// TIA Portal project "AutoII-G1" (V16)

(* hardware
DEVICE "S7-1200 station_1"  S7-1200 Station
   slot 0: "Rack_0"  S7-1200 Rack  Rack  V1.0
   slot 1: "PLC_1"  CPU 1214C DC/DC/DC  6ES7 214-1AG40-0XB0  V4.4
   slot 2: "DI 16/DQ 16x24VDC_1"  6ES7 223-1BL32-0XB0  V2.0
DEVICE "HMI_1"  KTP700 Basic PN
   slot 0: "HMI_1"  KTP700 Basic PN  6AV2 123-2GB03-0AX0  16.0.0.0
   slot 1: "HMI_RT_1"  KTP700 Basic PN  6AV2 123-2GB03-0AX0  16.0.0.0
   slot 5: "HMI_1.IE_CP_1"  PROFINET Interface  16.0.0.0
      slot 1: "Interfaz PROFINET_1"  PROFINET Interface
         slot 1: "Port_1"  Port
*)

// ===== PLC "PLC_1"  CPU 1214C DC/DC/DC =====

VAR_GLOBAL   // PLC tag table "Tabla de variables estándar"
   "ARRANQUE_M1" AT %I0.0 : Bool;
   "PARO_M1" AT %I0.1 : Bool;
   "FALLA_M1" AT %I0.2 : Bool;
   "MOTOR1" AT %Q0.0 : Bool;
   "ARRANQUE_M2" AT %I0.3 : Bool;
   "PARO_M2" AT %I0.4 : Bool;
   "FALLA_M2" AT %I0.5 : Bool;
   "MOTOR2" AT %Q0.1 : Bool;
   "ARRANQUE_M3" AT %I0.6 : Bool;
   "PARO_M3" AT %I0.7 : Bool;
   "FALLA_M3" AT %I1.0 : Bool;
   "MOTOR3" AT %Q0.2 : Bool;
   "Tag_1" AT %M0.0 : Bool;
   "Tag_2" AT %M0.1 : Bool;
   "Tag_3" AT %M0.2 : Bool;
   "Abrir_V1" AT %I2.0 : Bool;
   "Cerrar_V1" AT %I2.1 : Bool;
   "Q_Abrir_V1" AT %Q2.0 : Bool;
   "Aux_V1" AT %M2.0 : Bool;
   "Tag_4" AT %Q0.3 : Bool;
   "Conf_Ab_V1" AT %I2.2 : Bool;
   "Conf_Cer_V1" AT %I2.3 : Bool;
   "Q_Cerrar_V1" AT %Q2.1 : Bool;
   "HMI_Arranque_Secuencia" AT %M1.0 : Bool;
   "HMI_Paro_Secuencia" AT %M1.1 : Bool;
   "Reset_Fallas" AT %I2.4 : Bool;
   "Alarmas_1" AT %MW10 : Word;
   "Tag_5" AT %I3.0 : Bool;
   "Tag_6" AT %I3.1 : Bool;
   "Tag_7" AT %I3.3 : Bool;
   "Tag_8" AT %I3.2 : Bool;
   "Tag_9" AT %Q3.0 : Bool;
   "Tag_10" AT %Q3.1 : Bool;
   "Tag_11" AT %I4.0 : Bool;
   "Tag_12" AT %I4.1 : Bool;
   "Tag_13" AT %Q4.0 : Bool;
   "Tag_14" AT %Q4.1 : Bool;
   "LT-T001" AT %MD20 : Real;
   "SEÑAL T001" AT %MW18 : Int;
END_VAR

DATA_BLOCK "VALVULA_V1"   // DB3
{ S7_Optimized_Access := 'TRUE' }
VERSION : 0.1
// stored: InstanceOfName VALVULA
"VALVULA"
BEGIN
END_DATA_BLOCK

DATA_BLOCK "VALVULA_2"   // DB4
{ S7_Optimized_Access := 'TRUE' }
VERSION : 0.1
// stored: InstanceOfName VALVULA
"VALVULA"
BEGIN
END_DATA_BLOCK

DATA_BLOCK "VALVULA_3"   // DB5
{ S7_Optimized_Access := 'TRUE' }
VERSION : 0.1
// stored: InstanceOfName VALVULA
"VALVULA"
BEGIN
END_DATA_BLOCK

// folder: System blocks/Program resources

DATA_BLOCK "T_ON_M2"   // DB1
{ S7_Optimized_Access := 'TRUE' }
AUTHOR : Simatic
FAMILY : IEC
NAME : IEC_TMR
VERSION : 1.0
// stored: InstanceOfName IEC_TIMER
"IEC_TIMER"
BEGIN
END_DATA_BLOCK

DATA_BLOCK "T_ON_M3"   // DB2
{ S7_Optimized_Access := 'TRUE' }
AUTHOR : Simatic
FAMILY : IEC
NAME : IEC_TMR
VERSION : 1.0
// stored: InstanceOfName IEC_TIMER
"IEC_TIMER"
BEGIN
END_DATA_BLOCK

// folder: (top level)

FUNCTION_BLOCK "VALVULA"   // FB1, LAD
{ S7_Optimized_Access := 'TRUE' }
VERSION : 0.1
   VAR_INPUT
      Abrir : Bool;
      Conf_Abierta : Bool;
      Hab_Conf_Ab : Bool;
      T_Abrir : Time;
      T_Mon_Abrir : Time;
      Cerrar : Bool;
      Conf_Cerrada : Bool;
      Hab_Conf_Cer : Bool;
      T_Cierre : Time;
      T_Mon_Cierre : Time;
      Reset : Bool;
   END_VAR
   VAR_OUTPUT
      Q_Abrir : Bool;
      Q_Cerrar : Bool;
      Error_Abrir : Bool;
      Error_Cerrar : Bool;
   END_VAR
   VAR
      Aux_Valvula : Bool;
      Aux_Valvula2 : Bool;
      TP_Cierre : IEC_TIMER;
      TP_Abrir : IEC_TIMER;
      Mon_Abrir : IEC_TIMER;
      Mon_Cerrar : IEC_TIMER;
   END_VAR
BEGIN

REGION Network 1
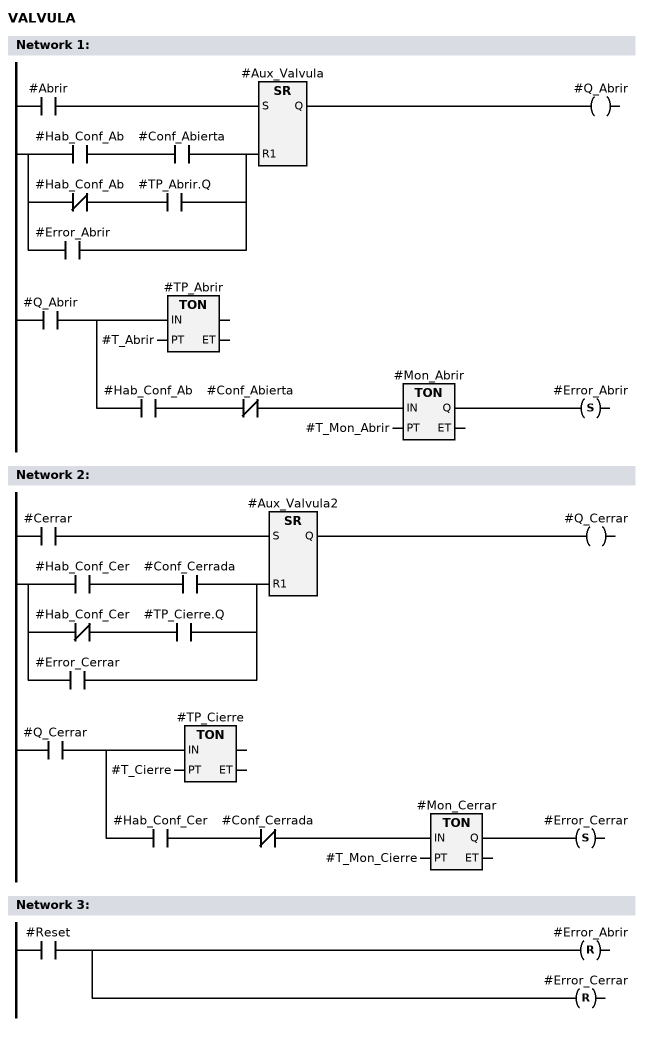
   IF #Abrir THEN
       #Aux_Valvula := TRUE;   // SR flip-flop
   END_IF;
   IF (#Hab_Conf_Ab AND #Conf_Abierta) OR (NOT #Hab_Conf_Ab AND #TP_Abrir.Q) OR #Error_Abrir THEN
       #Aux_Valvula := FALSE;
   END_IF;
   #Q_Abrir := #Aux_Valvula;
   #TP_Abrir.TON(IN := #Q_Abrir, PT := #T_Abrir);
   #Mon_Abrir.TON(IN := #Q_Abrir AND #Hab_Conf_Ab AND NOT #Conf_Abierta, PT := #T_Mon_Abrir);
   IF #Mon_Abrir.Q THEN #Error_Abrir := TRUE; END_IF;
END_REGION

REGION Network 2
   IF #Cerrar THEN
       #Aux_Valvula2 := TRUE;   // SR flip-flop
   END_IF;
   IF (#Hab_Conf_Cer AND #Conf_Cerrada) OR (NOT #Hab_Conf_Cer AND #TP_Cierre.Q) OR #Error_Cerrar THEN
       #Aux_Valvula2 := FALSE;
   END_IF;
   #Q_Cerrar := #Aux_Valvula2;
   #TP_Cierre.TON(IN := #Q_Cerrar, PT := #T_Cierre);
   #Mon_Cerrar.TON(IN := #Q_Cerrar AND #Hab_Conf_Cer AND NOT #Conf_Cerrada, PT := #T_Mon_Cierre);
   IF #Mon_Cerrar.Q THEN #Error_Cerrar := TRUE; END_IF;
END_REGION

REGION Network 3
   RUNG wire#powerrail
      Contact( #Reset )
      wire#w1
      R_Coil( #Error_Abrir )
   END_RUNG
   RUNG wire#w1
      R_Coil( #Error_Cerrar )
   END_RUNG
   // the same network as SCL:
   IF #Reset THEN
       #Error_Abrir := FALSE;
       #Error_Cerrar := FALSE;
   END_IF;
END_REGION
END_FUNCTION_BLOCK

FUNCTION "MOTOR" : Void   // FC1, LAD
{ S7_Optimized_Access := 'TRUE' }
VERSION : 0.1
   VAR_INPUT
      ARRANQUE : Bool;
      PARO : Bool;
      FALLA : Bool;
   END_VAR
   VAR_OUTPUT
      MOTOR : Bool;
   END_VAR
   VAR_IN_OUT
      mARRANQUE : Bool;
   END_VAR
BEGIN

REGION Network 1
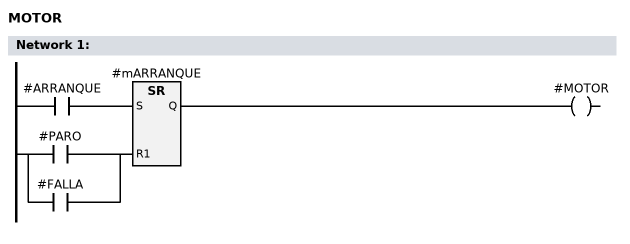
   RUNG wire#powerrail
      Contact( #ARRANQUE )
      S_SR(operand := #mARRANQUE, r1 := wire#w1)
      Coil( #MOTOR )
   END_RUNG
   RUNG wire#powerrail
      Contact( #PARO )
   END_RUNG wire#w1
   RUNG wire#powerrail
      Contact( #FALLA )
   END_RUNG wire#w1
   // the same network as SCL:
   IF #ARRANQUE THEN
       #mARRANQUE := TRUE;   // SR flip-flop
   END_IF;
   IF #PARO OR #FALLA THEN #mARRANQUE := FALSE; END_IF;
   #MOTOR := #mARRANQUE;
END_REGION
END_FUNCTION

FUNCTION "ESCALA" : Void   // FC2, LAD
{ S7_Optimized_Access := 'TRUE' }
VERSION : 0.1
   VAR_INPUT
      ENTRADA : Int;
      MIN_ENT : Int;
      MAX_ENT : Int;
      MIN_SAL : Real;
      MAX_SAL : Real;
   END_VAR
   VAR_OUTPUT
      VALOR : Real;
   END_VAR
   VAR_TEMP
      NORM : Real;
   END_VAR
BEGIN

REGION Network 1
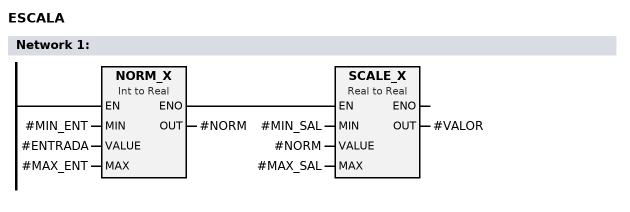
   RUNG wire#powerrail
      { S7_Templates := "[SrcType := Int, DestType := Real]" } Normalize(min := #MIN_ENT, value := #ENTRADA, max := #MAX_ENT, out => #NORM)
      { S7_Templates := "[SrcType := Real, DestType := Real]" } Scale(min := #MIN_SAL, value := #NORM, max := #MAX_SAL, out => #VALOR)
   END_RUNG
   // the same network as SCL:
   #NORM := NORM_X(MIN := #MIN_ENT, VALUE := #ENTRADA, MAX := #MAX_ENT);
   #VALOR := SCALE_X(MIN := #MIN_SAL, VALUE := #NORM, MAX := #MAX_SAL);
END_REGION
END_FUNCTION

ORGANIZATION_BLOCK "Main"   // OB1, LAD, ProgramCycle
TITLE = "Main Program Sweep (Cycle)"
{ S7_Optimized_Access := 'TRUE' }
VERSION : 0.1
BEGIN

REGION Network 1
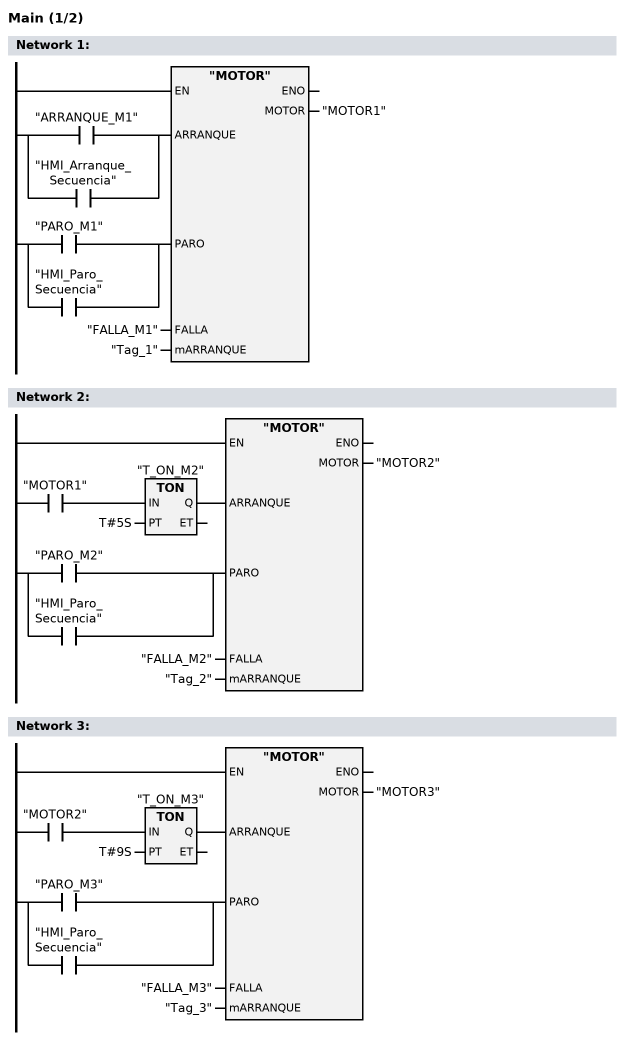
   RUNG wire#powerrail
      "MOTOR"(ARRANQUE := wire#w1, PARO := wire#w2, FALLA := "FALLA_M1", mARRANQUE := "Tag_1", MOTOR => "MOTOR1")
   END_RUNG
   RUNG wire#powerrail
      Contact( "ARRANQUE_M1" )
   END_RUNG wire#w1
   RUNG wire#powerrail
      Contact( "HMI_Arranque_Secuencia" )
   END_RUNG wire#w1
   RUNG wire#powerrail
      Contact( "PARO_M1" )
   END_RUNG wire#w2
   RUNG wire#powerrail
      Contact( "HMI_Paro_Secuencia" )
   END_RUNG wire#w2
   // the same network as SCL:
   "MOTOR"(ARRANQUE := "ARRANQUE_M1" OR "HMI_Arranque_Secuencia",
           PARO := "PARO_M1" OR "HMI_Paro_Secuencia",
           FALLA := "FALLA_M1",
           mARRANQUE := "Tag_1",
           MOTOR => "MOTOR1");
END_REGION

REGION Network 2
   "T_ON_M2".TON(IN := "MOTOR1", PT := T#5S);
   "MOTOR"(ARRANQUE := "T_ON_M2".Q,
           PARO := "PARO_M2" OR "HMI_Paro_Secuencia",
           FALLA := "FALLA_M2",
           mARRANQUE := "Tag_2",
           MOTOR => "MOTOR2");
END_REGION

REGION Network 3
   "T_ON_M3".TON(IN := "MOTOR2", PT := T#9S);
   "MOTOR"(ARRANQUE := "T_ON_M3".Q,
           PARO := "PARO_M3" OR "HMI_Paro_Secuencia",
           FALLA := "FALLA_M3",
           mARRANQUE := "Tag_3",
           MOTOR => "MOTOR3");
END_REGION

REGION Network 4
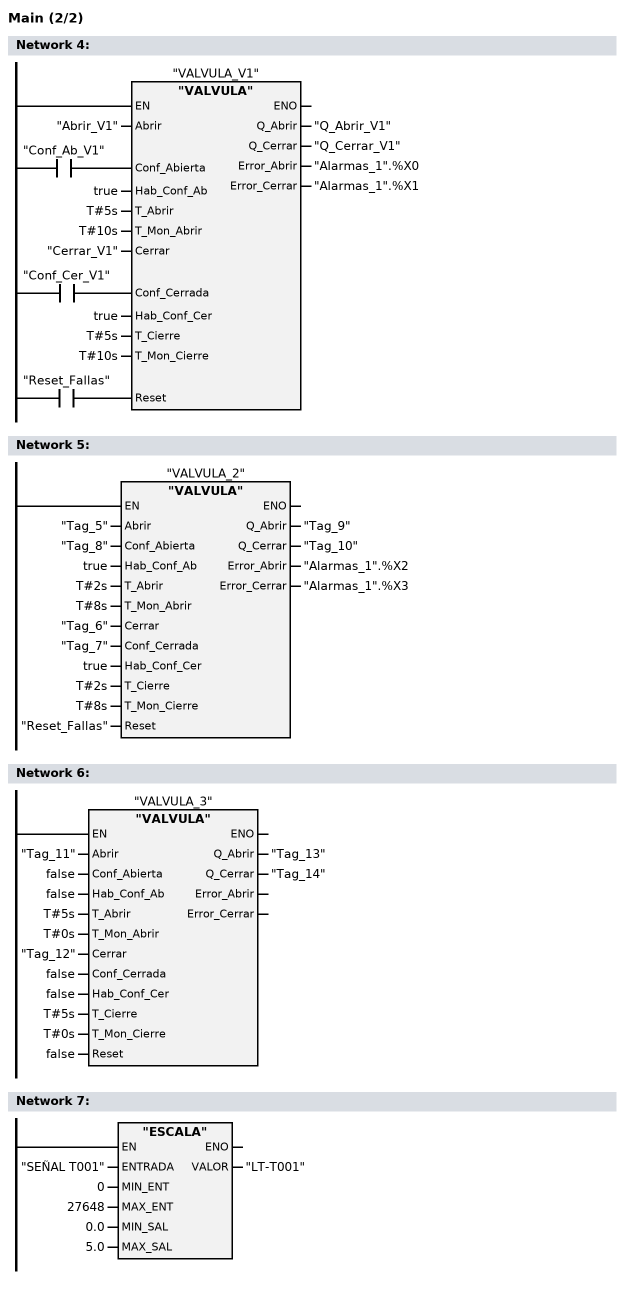
   RUNG wire#powerrail
      "VALVULA_V1"(Conf_Abierta := wire#w1, Conf_Cerrada := wire#w2, Reset := wire#w3, Abrir := "Abrir_V1", Hab_Conf_Ab := true, T_Abrir := T#5s, T_Mon_Abrir := T#10s, Cerrar := "Cerrar_V1", Hab_Conf_Cer := true, T_Cierre := T#5s, T_Mon_Cierre := T#10s, Q_Abrir => "Q_Abrir_V1", Q_Cerrar => "Q_Cerrar_V1", Error_Abrir => "Alarmas_1".%X0, Error_Cerrar => "Alarmas_1".%X1)
   END_RUNG
   RUNG wire#powerrail
      Contact( "Conf_Ab_V1" )
   END_RUNG wire#w1
   RUNG wire#powerrail
      Contact( "Conf_Cer_V1" )
   END_RUNG wire#w2
   RUNG wire#powerrail
      Contact( "Reset_Fallas" )
   END_RUNG wire#w3
   // the same network as SCL:
   "VALVULA_V1"(Abrir := "Abrir_V1",   // "VALVULA"
                Conf_Abierta := "Conf_Ab_V1",
                Hab_Conf_Ab := true,
                T_Abrir := T#5s,
                T_Mon_Abrir := T#10s,
                Cerrar := "Cerrar_V1",
                Conf_Cerrada := "Conf_Cer_V1",
                Hab_Conf_Cer := true,
                T_Cierre := T#5s,
                T_Mon_Cierre := T#10s,
                Reset := "Reset_Fallas",
                Q_Abrir => "Q_Abrir_V1",
                Q_Cerrar => "Q_Cerrar_V1",
                Error_Abrir => "Alarmas_1".%X0,
                Error_Cerrar => "Alarmas_1".%X1);
END_REGION

REGION Network 5
   RUNG wire#powerrail
      "VALVULA_2"(Abrir := "Tag_5", Conf_Abierta := "Tag_8", Hab_Conf_Ab := true, T_Abrir := T#2s, T_Mon_Abrir := T#8s, Cerrar := "Tag_6", Conf_Cerrada := "Tag_7", Hab_Conf_Cer := true, T_Cierre := T#2s, T_Mon_Cierre := T#8s, Reset := "Reset_Fallas", Q_Abrir => "Tag_9", Q_Cerrar => "Tag_10", Error_Abrir => "Alarmas_1".%X2, Error_Cerrar => "Alarmas_1".%X3)
   END_RUNG
   // the same network as SCL:
   "VALVULA_2"(Abrir := "Tag_5",   // "VALVULA"
               Conf_Abierta := "Tag_8",
               Hab_Conf_Ab := true,
               T_Abrir := T#2s,
               T_Mon_Abrir := T#8s,
               Cerrar := "Tag_6",
               Conf_Cerrada := "Tag_7",
               Hab_Conf_Cer := true,
               T_Cierre := T#2s,
               T_Mon_Cierre := T#8s,
               Reset := "Reset_Fallas",
               Q_Abrir => "Tag_9",
               Q_Cerrar => "Tag_10",
               Error_Abrir => "Alarmas_1".%X2,
               Error_Cerrar => "Alarmas_1".%X3);
END_REGION

REGION Network 6
   RUNG wire#powerrail
      "VALVULA_3"(Abrir := "Tag_11", Conf_Abierta := false, Hab_Conf_Ab := false, T_Abrir := T#5s, T_Mon_Abrir := T#0s, Cerrar := "Tag_12", Conf_Cerrada := false, Hab_Conf_Cer := false, T_Cierre := T#5s, T_Mon_Cierre := T#0s, Reset := false, Q_Abrir => "Tag_13", Q_Cerrar => "Tag_14", Error_Abrir =>, Error_Cerrar =>)
   END_RUNG
   // the same network as SCL:
   "VALVULA_3"(Abrir := "Tag_11",   // "VALVULA"
               Conf_Abierta := false,
               Hab_Conf_Ab := false,
               T_Abrir := T#5s,
               T_Mon_Abrir := T#0s,
               Cerrar := "Tag_12",
               Conf_Cerrada := false,
               Hab_Conf_Cer := false,
               T_Cierre := T#5s,
               T_Mon_Cierre := T#0s,
               Reset := false,
               Q_Abrir => "Tag_13",
               Q_Cerrar => "Tag_14");
END_REGION

REGION Network 7
   RUNG wire#powerrail
      "ESCALA"(ENTRADA := "SEÑAL T001", MIN_ENT := 0, MAX_ENT := 27648, MIN_SAL := 0.0, MAX_SAL := 5.0, VALOR => "LT-T001")
   END_RUNG
   // the same network as SCL:
   "ESCALA"(ENTRADA := "SEÑAL T001",
            MIN_ENT := 0,
            MAX_ENT := 27648,
            MIN_SAL := 0.0,
            MAX_SAL := 5.0,
            VALOR => "LT-T001");
END_REGION
END_ORGANIZATION_BLOCK

(* ===== HMI "HMI_RT_1" =====
system functions are stored by id; their names below are inferred from use
connection "HMI_Conexión_1": ETHERNET, SMART_S7_1200_OMS

HMI tags "Tabla de variables estándar"
   "HMI_Arranque_Secuencia" : Bool = PLC HMI_Arranque_Secuencia AT %M1.0, 1 s
   "HMI_Paro_Secuencia" : Bool = PLC HMI_Paro_Secuencia AT %M1.1, 1 s
   "MOTOR1" : Bool = PLC MOTOR1 AT %Q0.0, 1 s
   "MOTOR2" : Bool = PLC MOTOR2 AT %Q0.1, 1 s
   "MOTOR3" : Bool = PLC MOTOR3 AT %Q0.2, 1 s
   "Alarmas_1" : Word = PLC Alarmas_1 AT %MW10, 1 s
   "LT-T001" : Real = PLC "LT-T001" AT %MD20, 1 s

discrete alarms
   2: 'Falla de confirmación de cierre de válvula V1', class Errors, trigger "Alarmas_1" bit 1
   1: 'Falla de confirmación de apertura de válvula V1 / Falla relacionada con la ausencia de confirmación de apertura de la válvula Posibles causas: Falla en el suministro de aire comprimido. Falla en el sensor inductivo de detección de apertura.', class Errors, trigger "Alarmas_1" bit 0
   4: 'Falla de confirmación de cierre de válvula V2', class Errors, trigger "Alarmas_1" bit 3
   3: 'Falla de confirmación de apertura de válvula V2', class Errors, trigger "Alarmas_1" bit 2

analog alarms
   1: 'ALTO NIVEL EN TANQUE T001. LÍMITE 4,58 m ; VALOR ACTUAL', class Errors, trigger "LT-T001"
   2: 'BAJO NIVEL EN TANQUE T001. LÍMITE 0,52 m ; VALOR ACTUAL', class Errors, trigger "LT-T001"

Template "Plantilla_1" 800x480
   Button "Salir" at 714,429 size 71x50; TextOff 'Salir'; PictureOff "ExitRuntime_KTP700_Basic_PN_TR"; PictureOn "ExitRuntime_KTP700_Basic_PN_TR"
      on Release: StopRuntime(0)
   Button "Template_Button" at 614,429 size 71x50; TextOff 'Text'
   Button "Template_Button_1" at 514,429 size 71x50; TextOff 'Text'
   Button "Template_Button_2" at 414,429 size 71x50; TextOff 'Text'
   Button "Avisos" at 314,429 size 71x50; TextOff 'Avisos'; PictureOff "AlarmDisplay_KTP700_Basic_PN_TR"; PictureOn "AlarmDisplay_KTP700_Basic_PN_TR"
      on Release: function_ef3f5d25("Ventana de avisos_no_acusado", -1)
   Button "Template_Button_3" at 214,429 size 71x50; TextOff 'Text'
   Button "Template_Button_4" at 114,429 size 71x50; TextOff 'Text'
   Button "Imagen inicial" at 14,429 size 71x50; TextOff 'Imagen inicial'; PictureOff "NavigateHome_KTP700_Basic_PN_TR"; PictureOn "NavigateHome_KTP700_Basic_PN_TR"
      on Release: ActivateScreen("Principal", 0)

screen "Principal" 800x480, template "Plantilla_1"
   GraphicView "Visor de gráficos_1" at 0,62 size 799x355; Picture "horno"
   Button "Botón_1" at 65,9 size 95x45; TextOff 'ON'
      on Press: function_b14e0dd5("HMI_Arranque_Secuencia", 0)
   Button "Botón_2" at 664,9 size 95x45; TextOff 'OFF'
      on Press: function_b14e0dd5("HMI_Paro_Secuencia", 0)
   Circle "Círculo_1" at 131,136 size 39x39
      Appearance <- "MOTOR1"
   Circle "Círculo_2" at 391,130 size 39x39
      Appearance <- "MOTOR2"
   Circle "Círculo_3" at 631,125 size 39x39
      Appearance <- "MOTOR3"
*)